(* Logix 5000 project; controller IoT 1756-L85E rev 33.12; software revision 33.01 *)

TASK MainTask (continuous, watchdog 500 ms) : MainProgram

MODULES
   Local : 1756-L85E (ICP 0, rev 33.12)
      Ethernet_IP : 1756-EN2T (ICP 1, Ethernet 172.17.99.2, rev 11.2, Input RPI 500 ms)
END_MODULES

VAR_GLOBAL   (* controller tags *)
   frequency : REAL := 1.0;
   Function : REAL := 43.87703;
   IoT_data : DINT := 44;
   time_index : REAL := 214.1288;
END_VAR

PROGRAM MainProgram   (* main routine MainRoutine *)
VAR
   sample_time : TIMER := (PRE := 100, ACC := 100, EN := 1, DN := 1);
END_VAR

ROUTINE MainRoutine   (* ladder *)
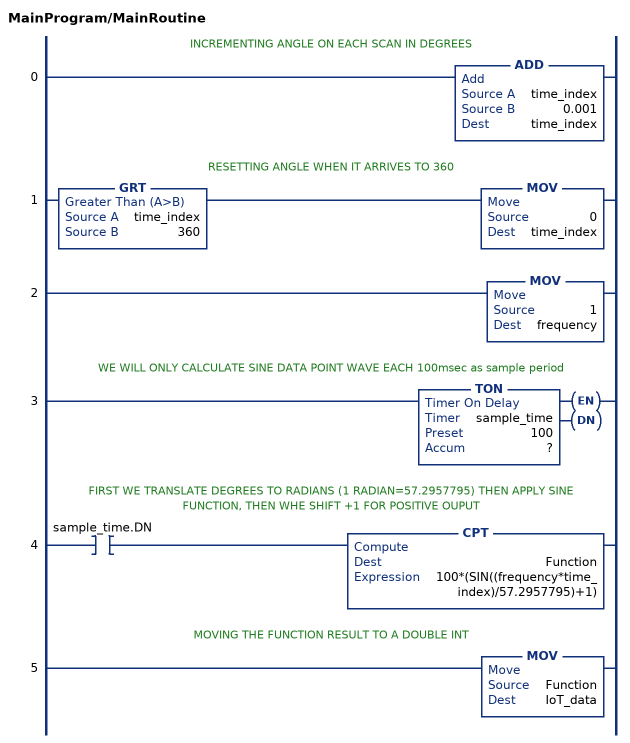
   // INCREMENTING ANGLE ON EACH SCAN IN DEGREES
   0: ADD(time_index,0.001,time_index);
   // RESETTING ANGLE WHEN IT ARRIVES TO 360
   1: GRT(time_index,360)MOV(0,time_index);
   2: MOV(1,frequency);
   // WE WILL ONLY CALCULATE SINE DATA POINT WAVE EACH 100msec as sample period
   3: TON(sample_time,?,?);
   // FIRST WE TRANSLATE DEGREES TO RADIANS (1 RADIAN=57.2957795) THEN APPLY SINE FUNCTION, THEN WHE SHIFT +1 FOR POSITIVE OUPUT
   4: XIC(sample_time.DN)CPT(Function,100*(SIN((frequency*time_index)/57.2957795)+1));
   // MOVING THE FUNCTION RESULT TO A DOUBLE INT
   5: MOV(Function,IoT_data);
END_ROUTINE
END_PROGRAM
